// TwinCAT 3 PLC project PLC1
// ProgramVersion: 3.1.4024.0
// libraries:
//   Tc2_Standard, * (Beckhoff Automation GmbH)
//   Tc2_System, * (Beckhoff Automation GmbH)
//   Tc3_Module, * (Beckhoff Automation GmbH)
//   VisuSymbols,3.5.10.0,System
// project tree:
//   / GlobalTextList.TcGTLO, PlcTask.TcTTO, Visualization Manager.TcVMO (not stored)
//   GVLs/ GVL.TcGVL
//   POUs/ FC1_Bereken_Snelheid.TcPOU, MAIN.TcPOU, POU.TcPOU, PRG1_Conveyer_Operation.TcPOU, PRG2_Object_Detection.TcPOU
//   VISUs/ Visu_gewicht_en_snelheid.TcVIS

CONFIGURATION PLC1
    RESOURCE PLC ON TwinCAT3
        TASK PlcTask(INTERVAL := T#10ms, PRIORITY := 20);
        PROGRAM MAIN WITH PlcTask : MAIN;
    END_RESOURCE
END_CONFIGURATION

// ---- GVLs/GVL.TcGVL
{attribute 'qualified_only'}
VAR_GLOBAL

// Hele rits aan variabelen

// -----------------------------------------Ingangen	
// Digitale Ingangen
	In0Res AT%IB00 : BOOL := 0;  //Reserve
	In1Res AT%IB01 : BOOL := 0;  //Reserve
	In2Res AT%IB02 : BOOL := 0;  //Reserve
	In3Res AT%IB03 : BOOL := 0;  //Reserve 
	In4Res AT%IB04 : BOOL := 0;  //Reserve 
	In5Res AT%IB05 : BOOL := 0;  //Reserve 
	In6Res AT%IB06 : BOOL := 0;  //Reserve
	In7Res AT%IB07 : BOOL := 0;  //Reserve 
	In8Res AT%IB08 : BOOL := 0;  //Reserve 
	In9Res AT%IB09 : BOOL := 0;  //Reserve
	
// Analoge ingangen 
	weegcelWaarde AT%IW10 : DINT := 0;  //ingelezen gewicht van de lading 
	In11Res AT%IW11 : DINT := 0;  //Reserve 
	In12Res AT%IW12 : DINT := 0;  //Reserve 
	In13Res AT%IW13 : DINT := 0;  //Reserve 
	In14Res AT%IW14 : DINT := 0;  //Reserve 
	In15Res AT%IW15 : DINT := 0;  //Reserve 
	In16Res AT%IW16 : DINT := 0;  //Reserve
	In17Res AT%IW17 : DINT := 0;  //Reserve
	In18Res AT%IW18 : DINT := 0;  //Reserve
	In19Res AT%IW19 : DINT := 0;  //Reserve
	
// -----------------------------------------Uitgangen
// Digitale Uitgangen
	Uit0Res AT%QB00 : BOOL := 0;  //Reserve
	Uit1Res AT%QB01 : BOOL := 0;  //Reserve 
	Uit2Res AT%QB02 : BOOL := 0;  //Reserve
	Uit3Res AT%QB03 : BOOL := 0;  //Reserve
	Uit4Res AT%QB04 : BOOL := 0;  //Reserve
	Uit5Res AT%QB05 : BOOL := 0;  //Reserve
	Uit6Res AT%QB06 : BOOL := 0;  //Reserve
	Uit7Res AT%QB07 : BOOL := 0;  //Reserve
	Uit8Res AT%QB08 : BOOL := 0;  //Reserve
	Uit9Res AT%QB09 : BOOL := 0;  //Reserve
	
// Analoge Uitgangen 
	geschrevenSnelheid AT%QW10 : DINT := 0;  // snelheid uitgeschreven naar motor
	Uit11Res AT%QW11 : DINT := 0;  //Reserve
	Uit12Res AT%QW12 : DINT := 0;  //Reserve
	Uit13Res AT%QW13 : DINT := 0;  //Reserve
	Uit14Res AT%QW14 : DINT := 0;  //Reserve
	Uit15Res AT%QW15 : DINT := 0;  //Reserve
	Uit16Res AT%QW16 : DINT := 0;  //Reserve
	Uit17Res AT%QW17 : DINT := 0;  //Reserve
	Uit18Res AT%QW18 : DINT := 0;  //Reserve 
	Uit19Res AT%QW19 : DINT := 0;  //Reserve


// Globale Variabelen
	ladingGewicht AT%MW10 : DINT := 0; //opslag gelezen gewicht 

END_VAR

// ---- POUs/MAIN.TcPOU
PROGRAM MAIN
VAR
END_VAR


// Call Programs
PRG1_Conveyer_Operation();
PRG2_Object_Detection();

END_PROGRAM

// ---- POUs/PRG1_Conveyer_Operation.TcPOU
PROGRAM PRG1_Conveyer_Operation
VAR
END_VAR


// bereken snelheid

GVL.ladingGewicht := GVL.weegcelWaarde;									
GVL.geschrevenSnelheid := FC1_Bereken_Snelheid(GVL.ladingGewicht);

END_PROGRAM

// ---- POUs/FC1_Bereken_Snelheid.TcPOU
FUNCTION FC1_Bereken_Snelheid : DINT
VAR_INPUT
	gelezenGewicht : DINT := 0;
END_VAR
VAR
	mid : DINT := 0;
	berekendeSnelheid : DINT := 0;
END_VAR


mid := gelezenGewicht / 5;
berekendeSnelheid := mid * 6;

END_FUNCTION

// ---- POUs/PRG2_Object_Detection.TcPOU
PROGRAM PRG2_Object_Detection
VAR
END_VAR

END_PROGRAM

// ---- POUs/POU.TcPOU


// ---- VISUs/Visu_gewicht_en_snelheid.TcVIS
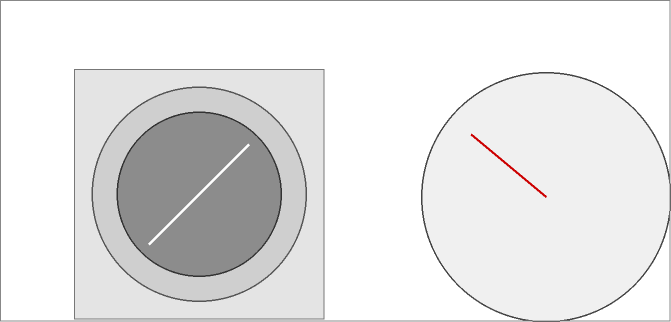
VISUALIZATION Visu_gewicht_en_snelheid  // 671x322
    Meter180 (421,72 250x250), value: GVL.geschrevenSnelheid, style: Meter-Meter180-Gray, scale format: %.1f, scale 0..100
    Potentiometer360 (74,69 250x250), variable: GVL.ladingGewicht, style: Potentiometer-Potentiometer360-Gray, scale format: %.1f, scale 0..100
        p2431819421: Outside
END_VISUALIZATION
